FUNCTION_BLOCK visControl
VAR_INPUT
END_VAR
VAR_OUTPUT
END_VAR
VAR
	Idx : INT;
	nPrevIdx : INT;
END_VAR


Idx := GVL_visVariableMap.visValveMaskIdx;


IF GVL_visVariableMap.nValveMask <> 0 THEN
	GVL_visVariableMap.anValveMask[Idx] := GVL_visVariableMap.nValveMask;
	GVL_visVariableMap.nValveMask := 0; // To Clear the Text Box
END_IF

END_FUNCTION_BLOCK

(* stored: Version 1.1.0.1
   POU visControl: Id {44e419da-d1ca-0ad4-1138-0ce61d4d2251}, SpecialFunc None *)
